PROGRAM prgCS
VAR
	fbCS		: FB_ECS_Keba_P30;
	bEnableCS	: BOOL;
	lrPowerCS	: LREAL;
END_VAR
VAR PERSISTENT

END_VAR

fbCS(
	bEnable := bEnableCS,
	bPowerDataInvers := FALSE,
	byElectricFuseLine := 1,
	uiFailsafeCurrent := ,
	uiFailsafeTimeOut := ,
	diNrOfEMS_IN := ,
	diNrOfEM_IN_CS := ,
	sIPAdress := '192.168.178.51',
	stSetupECS := ,
	stDataECS => ,
	diNrOfECS_OUT => ,
	lrTotalPowerECSRealTime => lrPowerCS );

END_PROGRAM

(* stored: Version 1.1.0.1, ProductVersion 3.1.4024.9
   POU prgCS: Id {cf38982a-1a4e-4f90-87d5-58e8c65a1cce}, SpecialFunc None *)
